ABB RAPID module: Module1.mod

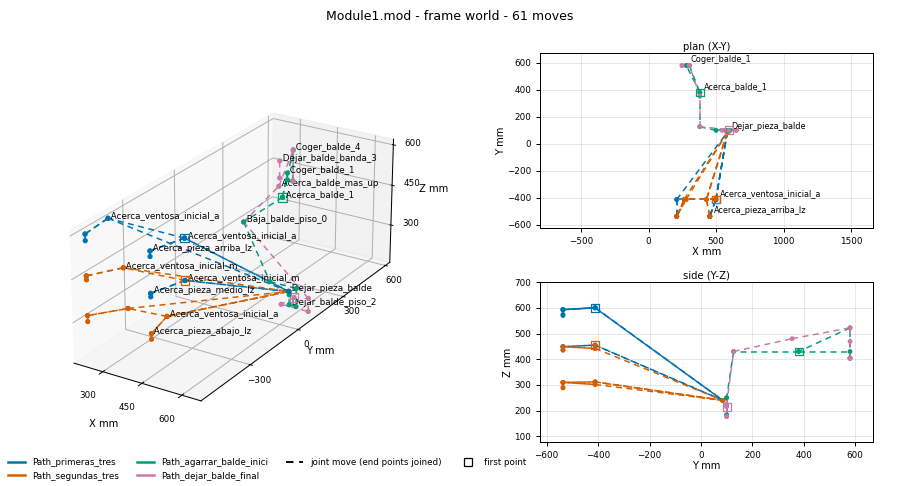
[picture p0: tool path of Module1.mod in frame world, 61 of 62 moves have a stored position in this frame; points joined in program order, loops and branches not executed]
MODULE Module1
    CONST jointtarget JointTarget_1:=[[0,0,0,0,0,0],[9E+09,9E+09,9E+09,9E+09,9E+09,9E+09]];
    CONST robtarget Acerca_balde:=[[100,70,-180],[1,0,0,0],[0,0,-1,0],[9E+09,9E+09,9E+09,9E+09,9E+09,9E+09]];
    CONST robtarget negativo_x_mundo_balde:=[[-100,170,-180],[1,0,0,0],[0,0,-1,0],[9E+09,9E+09,9E+09,9E+09,9E+09,9E+09]];
    CONST robtarget negativo_z_mundo_balde:=[[-100.000020105,169.99997294,-154.000005055],[1,0.000000007,-0.00000001,0.000000008],[0,0,-1,0],[9E+09,9E+09,9E+09,9E+09,9E+09,9E+09]];
    CONST robtarget positivo_x_mundo_balde:=[[-100,147,-154],[1,0,0,0],[0,0,-1,0],[9E+09,9E+09,9E+09,9E+09,9E+09,9E+09]];
    CONST robtarget positivo_z_mundo_balde:=[[-100,147,-217],[1,0,0,0],[0,0,-1,0],[9E+09,9E+09,9E+09,9E+09,9E+09,9E+09]];
    CONST robtarget Baja_balde_piso_0:=[[353,70,-180],[1,0,0,0],[0,0,-1,0],[9E+09,9E+09,9E+09,9E+09,9E+09,9E+09]];
    CONST robtarget Baja_balde_piso_1:=[[380,-50,0],[1,0,0,0],[0,0,-1,0],[9E+09,9E+09,9E+09,9E+09,9E+09,9E+09]];
    CONST robtarget Baja_balde_piso_2:=[[380.0000088,-152.999992201,0.000005224],[1,0.000000008,0,-0.000000022],[0,-1,-2,0],[9E+09,9E+09,9E+09,9E+09,9E+09,9E+09]];
    CONST robtarget negativo_z_balde_piso:=[[380,-153,67],[1,0,0,0],[0,0,0,0],[9E+09,9E+09,9E+09,9E+09,9E+09,9E+09]];
    CONST robtarget negativo_x_gancho_mundo_piso:=[[380,-126,67],[1,0,0,0],[0,0,-1,0],[9E+09,9E+09,9E+09,9E+09,9E+09,9E+09]];
    CONST robtarget positivo_z_gancho_mundo_piso:=[[380,-126,30],[1,0,0,0],[0,0,-1,0],[9E+09,9E+09,9E+09,9E+09,9E+09,9E+09]];
    CONST robtarget Diagonal_bajar_manija:=[[380,-185,60],[1,0,0,0],[0,0,-1,0],[9E+09,9E+09,9E+09,9E+09,9E+09,9E+09]];
    CONST robtarget Acerca_ventosa_inicial_arriba_Iz:=[[100,200,112],[1,0,0,0],[-1,-2,0,0],[9E+09,9E+09,9E+09,9E+09,9E+09,9E+09]];
    CONST robtarget negativ_y_vento_work_arriba_Iz:=[[145,75,122],[1,0,0,0],[-1,-2,0,0],[9E+09,9E+09,9E+09,9E+09,9E+09,9E+09]];
    CONST robtarget Dejar_pieza_en_balde:=[[-19.141559839,402.142254512,270],[1,0,0,-0.000000001],[-1,-2,0,0],[9E+09,9E+09,9E+09,9E+09,9E+09,9E+09]];
    CONST robtarget Acerca_ventosa_inicial_arriba_De:=[[390,200,111],[1,0,0,0],[-1,-2,0,0],[9E+09,9E+09,9E+09,9E+09,9E+09,9E+09]];
    CONST robtarget negativ_y_vento_work_arriba_De:=[[390,75,119],[1,0,0,0],[-1,-2,0,0],[9E+09,9E+09,9E+09,9E+09,9E+09,9E+09]];
    CONST robtarget Acerca_ventosa_inicial_medio_Iz:=[[100,200,257],[1,0,0,0],[-1,-2,0,0],[9E+09,9E+09,9E+09,9E+09,9E+09,9E+09]];
    CONST robtarget negativ_y_vento_work_medio_Iz:=[[145,75,258],[1,0,0,0],[-1,-2,0,0],[9E+09,9E+09,9E+09,9E+09,9E+09,9E+09]];
    CONST robtarget Agarrar_balde_again_ini:=[[380,-145,35],[1,0,0,0],[0,0,-1,0],[9E+09,9E+09,9E+09,9E+09,9E+09,9E+09]];
    CONST robtarget Agarrar_balde_again_z_nega_mun:=[[380.0000022,-95.000012886,73.00000505],[1,0.000000008,0,-0.000000022],[0,0,-2,0],[9E+09,9E+09,9E+09,9E+09,9E+09,9E+09]];
    CONST robtarget Agarrar_balde_again_x_posi_mun:=[[380,-200,73],[1,0,0,0],[0,0,-1,0],[9E+09,9E+09,9E+09,9E+09,9E+09,9E+09]];
    CONST robtarget Agarrar_balde_again_z_posi_mun:=[[380,-200,25],[1,0,0,0],[0,0,-1,0],[9E+09,9E+09,9E+09,9E+09,9E+09,9E+09]];
    CONST robtarget negativo_z_mundo_balde_dejar:=[[-100,147,-154],[1,0,0,0],[0,0,-1,0],[9E+09,9E+09,9E+09,9E+09,9E+09,9E+09]];
    CONST robtarget negativo_x_mundo_balde_dejar:=[[-100,202,-154],[1,0,0,0],[0,0,-1,0],[9E+09,9E+09,9E+09,9E+09,9E+09,9E+09]];
    CONST robtarget positivo_z_mundo_balde_dejar_H:=[[-100,202,-219],[1,0,0,0],[0,0,-1,0],[9E+09,9E+09,9E+09,9E+09,9E+09,9E+09]];
    CONST robtarget Acerca_ventosa_inicial_medio_De:=[[335,200,270],[1,0,0,0],[-1,-2,0,0],[9E+09,9E+09,9E+09,9E+09,9E+09,9E+09]];
    CONST robtarget negativ_y_vento_work_medio_De:=[[390,75,270],[1,0,0,0],[-1,-2,0,0],[9E+09,9E+09,9E+09,9E+09,9E+09,9E+09]];
    CONST robtarget Punto_intermedio_abajo_Iz:=[[170,200,300],[1,0,0,0],[-1,-2,0,0],[9E+09,9E+09,9E+09,9E+09,9E+09,9E+09]];
    CONST robtarget Acerca_ventosa_inicial_abajo_Iz:=[[170,200,400],[1,0,0,0],[-1,-2,0,0],[9E+09,9E+09,9E+09,9E+09,9E+09,9E+09]];
    CONST robtarget negativ_y_vento_work_abajo_Iz_3:=[[145,75,412],[1,0,0,0],[-1,-2,0,0],[9E+09,9E+09,9E+09,9E+09,9E+09,9E+09]];
    CONST robtarget Acerca_ventosa_inicial_abajo_De:=[[320,200,410],[1,0,0,0],[-1,-2,0,0],[9E+09,9E+09,9E+09,9E+09,9E+09,9E+09]];
    CONST robtarget negativ_y_vento_work_abajo_De_3:=[[390,75,412],[1,0,0,0],[-1,-2,0,0],[9E+09,9E+09,9E+09,9E+09,9E+09,9E+09]];
    CONST robtarget Acerca_pieza_arriba_Iz:=[[145,75,119],[1,0,0,0],[-1,-2,0,0],[9E+09,9E+09,9E+09,9E+09,9E+09,9E+09]];
    CONST robtarget Tomar_pieza_arriba_De:=[[390,75,141.8],[1,0,0,0],[-1,-2,0,0],[9E+09,9E+09,9E+09,9E+09,9E+09,9E+09]];
    CONST robtarget Tomar_pieza_medio_Iz:=[[145,75,275],[1,0,0,0],[-1,-2,0,0],[9E+09,9E+09,9E+09,9E+09,9E+09,9E+09]];
    CONST robtarget Tomar_pieza_arriba_Iz:=[[145,75,137.7],[1,0,0,0],[-1,-2,0,0],[9E+09,9E+09,9E+09,9E+09,9E+09,9E+09]];
    CONST robtarget Dejar_pieza_balde:=[[20,-15,-240],[1,0,0,0],[0,-1,0,0],[9E+09,9E+09,9E+09,9E+09,9E+09,9E+09]];
    CONST robtarget Acerca_pieza_arriba_De:=[[390,75,119],[1,0,0,0],[-1,-2,0,0],[9E+09,9E+09,9E+09,9E+09,9E+09,9E+09]];
    CONST robtarget Acerca_pieza_medio_Iz:=[[145,75,263],[1,0,0,0],[-1,-2,0,0],[9E+09,9E+09,9E+09,9E+09,9E+09,9E+09]];
    CONST robtarget Acerca_balde_mas_up:=[[125,70,-230],[1,0,0,0],[0,0,-1,0],[9E+09,9E+09,9E+09,9E+09,9E+09,9E+09]];
    CONST robtarget Tomar_pieza_medio_De:=[[390,75,276.9],[1,0,0,0],[-1,-2,0,0],[9E+09,9E+09,9E+09,9E+09,9E+09,9E+09]];
    CONST robtarget Tomar_pieza_abajo_De:=[[390,75,423.2],[1,0,0,0],[-1,-2,0,0],[9E+09,9E+09,9E+09,9E+09,9E+09,9E+09]];
    CONST robtarget Acerca_pieza_medio_De:=[[390,75,263],[1,0,0,0],[-1,-2,0,0],[9E+09,9E+09,9E+09,9E+09,9E+09,9E+09]];
    CONST robtarget Tomar_pieza_abajo_Iz:=[[145,75,421.6],[1,0,0,0],[-1,-2,0,0],[9E+09,9E+09,9E+09,9E+09,9E+09,9E+09]];
    CONST robtarget Acerca_pieza_abajo_Iz:=[[145,75,402],[1,0,0,0],[-1,-2,0,0],[9E+09,9E+09,9E+09,9E+09,9E+09,9E+09]];
    CONST robtarget Acerca_pieza_abajo_De:=[[390,75,402],[1,0,0,0],[-1,-2,0,0],[9E+09,9E+09,9E+09,9E+09,9E+09,9E+09]];
    CONST robtarget Acerca_balde_1:=[[100,70,-180],[1,0,0,0],[0,0,-1,0],[9E+09,9E+09,9E+09,9E+09,9E+09,9E+09]];
    CONST robtarget Coger_balde_1:=[[-100,170,-180],[1,0,0,0],[0,0,-1,0],[9E+09,9E+09,9E+09,9E+09,9E+09,9E+09]];
    CONST robtarget Coger_balde_2:=[[-100.000020105,169.99997294,-154.000005055],[1,0.000000007,-0.00000001,0.000000008],[0,0,-1,0],[9E+09,9E+09,9E+09,9E+09,9E+09,9E+09]];
    CONST robtarget Coger_balde_3:=[[-100,147,-154],[1,0,0,0],[0,0,-1,0],[9E+09,9E+09,9E+09,9E+09,9E+09,9E+09]];
    CONST robtarget Coger_balde_4:=[[-100,147,-272],[1,0,0,0],[0,0,-1,0],[9E+09,9E+09,9E+09,9E+09,9E+09,9E+09]];
    CONST robtarget Dejar_balde_piso_1:=[[380,-153,67],[1,0,0,0],[0,0,0,0],[9E+09,9E+09,9E+09,9E+09,9E+09,9E+09]];
    CONST robtarget Dejar_balde_piso_2:=[[380,-126,67],[1,0,0,0],[0,0,-1,0],[9E+09,9E+09,9E+09,9E+09,9E+09,9E+09]];
    CONST robtarget Dejar_balde_piso_3:=[[380,-126,30],[1,0,0,0],[0,0,-1,0],[9E+09,9E+09,9E+09,9E+09,9E+09,9E+09]];
    CONST robtarget Dejar_balde_banda_1:=[[-100,147,-154],[1,0,0,0],[0,0,-1,0],[9E+09,9E+09,9E+09,9E+09,9E+09,9E+09]];
    CONST robtarget Dejar_balde_banda_2:=[[-100,202,-154],[1,0,0,0],[0,0,-1,0],[9E+09,9E+09,9E+09,9E+09,9E+09,9E+09]];
    CONST robtarget Dejar_balde_banda_3:=[[-100,202,-219],[1,0,0,0],[0,0,-1,0],[9E+09,9E+09,9E+09,9E+09,9E+09,9E+09]];
    CONST robtarget Dejar_pieza_balde_2:=[[20,-15,-240],[0.707106781,0,0.707106781,0],[0,-1,-1,0],[9E+09,9E+09,9E+09,9E+09,9E+09,9E+09]];
    !***********************************************************
    !
    ! Módulo:  Module1
    !
    ! Descripción:
    !   <Introduzca la descripción aquí>
    !
    ! Autor: ASUS
    !
    ! Versión: 1.0
    !
    !***********************************************************


    !***********************************************************
    !
    ! Procedimiento Main
    !
    !   Este es el punto de entrada de su programa
    !
    !***********************************************************
    PROC main()
        !Añada aquí su código

        Home; !Inicio en Home
        Path_agarrar_balde_inicio;   !Coger balde de la banda y ponerlo en el piso
        Path_primeras_tres;   !Agarrar_primeras_tres_piezas
        !Path_segundas_tres;  !Agarrar_segundas_tres_piezas
        Path_dejar_balde_final;  !Dejar balde otra vez en la banda
        Home; !Finalizacion en Home

    ENDPROC

    PROC Home()
        MoveAbsJ JointTarget_1,v300,z100,Gancho\WObj:=Workobject_banda_gancho;
    ENDPROC
    PROC Path_primeras_tres()
        SetDO DO_01,0;
        SetDO DO_02,0;
        MoveJ Acerca_ventosa_inicial_arriba_Iz,v100,z100,Ventosa\WObj:=Workobject_Ventosa_Estante;
        SetDO DO_01,0;
        WaitTime 1;
        SetDO DO_02,1;
        WaitTime 1;
        MoveJ Acerca_pieza_arriba_Iz,v100,z100,Ventosa\WObj:=Workobject_Ventosa_Estante;
        MoveJ Tomar_pieza_arriba_Iz,v30,z100,Ventosa\WObj:=Workobject_Ventosa_Estante;
        MoveJ Acerca_pieza_arriba_Iz,v100,z100,Ventosa\WObj:=Workobject_Ventosa_Estante;
        MoveJ Acerca_ventosa_inicial_arriba_Iz,v100,z100,Ventosa\WObj:=Workobject_Ventosa_Estante;
        MoveJ Dejar_pieza_balde,v100,z100,Ventosa\WObj:=Workobject_Dejar_pieza_balde;
        WaitTime 1;
        SetDO DO_02,0;
        WaitTime 1;
        SetDO DO_01,1;
        WaitTime 1;
        MoveJ Acerca_ventosa_inicial_arriba_Iz,v100,z100,Ventosa\WObj:=Workobject_Ventosa_Estante;
        MoveJ Acerca_ventosa_inicial_arriba_De,v100,z100,Ventosa\WObj:=Workobject_Ventosa_Estante;
        WaitTime 1;
        SetDO DO_01,0;
        WaitTime 1;
        SetDO DO_02,1;
        WaitTime 1;
        MoveJ Acerca_pieza_arriba_De,v100,z100,Ventosa\WObj:=Workobject_Ventosa_Estante;
        MoveJ Tomar_pieza_arriba_De,v30,z100,Ventosa\WObj:=Workobject_Ventosa_Estante;
        MoveJ Acerca_pieza_arriba_De,v100,z100,Ventosa\WObj:=Workobject_Ventosa_Estante;
        MoveJ Acerca_ventosa_inicial_arriba_De,v100,z100,Ventosa\WObj:=Workobject_Ventosa_Estante;
        MoveJ Dejar_pieza_balde,v100,z100,Ventosa\WObj:=Workobject_Dejar_pieza_balde;
        WaitTime 1;
        SetDO DO_02,0;
        WaitTime 1;
        SetDO DO_01,1;
        WaitTime 1;
        MoveJ Acerca_ventosa_inicial_medio_Iz,v100,z100,Ventosa\WObj:=Workobject_Ventosa_Estante;
        WaitTime 1;
        SetDO DO_01,0;
        WaitTime 1;
        SetDO DO_02,1;
        WaitTime 1;
        MoveJ Acerca_pieza_medio_Iz,v100,z100,Ventosa\WObj:=Workobject_Ventosa_Estante;
        MoveJ Tomar_pieza_medio_Iz,v30,z100,Ventosa\WObj:=Workobject_Ventosa_Estante;
        MoveJ Acerca_pieza_medio_Iz,v100,z100,Ventosa\WObj:=Workobject_Ventosa_Estante;
        MoveJ Acerca_ventosa_inicial_medio_Iz,v100,z100,Ventosa\WObj:=Workobject_Ventosa_Estante;
        MoveJ Dejar_pieza_balde,v100,z100,Ventosa\WObj:=Workobject_Dejar_pieza_balde;
        WaitTime 1;
        SetDO DO_02,0;
        WaitTime 1;
        SetDO DO_01,1;
        WaitTime 1;
        SetDO DO_01,0;
        WaitTime 1;
    ENDPROC

    PROC Path_segundas_tres()
        MoveJ Acerca_ventosa_inicial_medio_Iz,v100,z100,Ventosa\WObj:=Workobject_Ventosa_Estante;
        MoveJ Acerca_ventosa_inicial_medio_De,v100,z100,Ventosa\WObj:=Workobject_Ventosa_Estante;
        WaitTime 1;
        SetDO DO_01,0;
        WaitTime 1;
        SetDO DO_02,1;
        WaitTime 1;
        MoveJ Acerca_pieza_medio_De,v100,z100,Ventosa\WObj:=Workobject_Ventosa_Estante;
        MoveJ Tomar_pieza_medio_De,v30,z100,Ventosa\WObj:=Workobject_Ventosa_Estante;
        MoveJ Acerca_pieza_medio_De,v100,z100,Ventosa\WObj:=Workobject_Ventosa_Estante;
        MoveJ Acerca_ventosa_inicial_medio_De,v100,z100,Ventosa\WObj:=Workobject_Ventosa_Estante;
        MoveJ Dejar_pieza_balde_2,v1000,z100,Ventosa\WObj:=Workobject_Dejar_pieza_balde_2;
        WaitTime 1;
        SetDO DO_02,0;
        WaitTime 1;
        SetDO DO_01,1;
        WaitTime 1;
        MoveJ Acerca_ventosa_inicial_abajo_Iz,v100,z100,Ventosa\WObj:=Workobject_Ventosa_Estante;
        WaitTime 1;
        SetDO DO_01,0;
        WaitTime 1;
        SetDO DO_02,1;
        WaitTime 1;
        MoveJ Acerca_pieza_abajo_Iz,v100,z100,Ventosa\WObj:=Workobject_Ventosa_Estante;
        MoveJ Tomar_pieza_abajo_Iz,v30,z100,Ventosa\WObj:=Workobject_Ventosa_Estante;
        MoveJ Acerca_pieza_abajo_Iz,v100,z100,Ventosa\WObj:=Workobject_Ventosa_Estante;
        MoveJ Acerca_ventosa_inicial_abajo_Iz,v100,z100,Ventosa\WObj:=Workobject_Ventosa_Estante;
        MoveJ Dejar_pieza_balde_2,v1000,z100,Ventosa\WObj:=Workobject_Dejar_pieza_balde_2;
        WaitTime 1;
        SetDO DO_02,0;
        WaitTime 1;
        SetDO DO_01,1;
        WaitTime 1;
        MoveJ Acerca_ventosa_inicial_abajo_Iz,v100,z100,Ventosa\WObj:=Workobject_Ventosa_Estante;
        MoveJ Acerca_ventosa_inicial_abajo_De,v100,z100,Ventosa\WObj:=Workobject_Ventosa_Estante;
        WaitTime 1;
        SetDO DO_01,0;
        WaitTime 1;
        SetDO DO_02,1;
        WaitTime 1;
        MoveJ Acerca_pieza_abajo_De,v100,z100,Ventosa\WObj:=Workobject_Ventosa_Estante;
        MoveJ Tomar_pieza_abajo_De,v30,z100,Ventosa\WObj:=Workobject_Ventosa_Estante;
        MoveJ Acerca_pieza_abajo_De,v100,z100,Ventosa\WObj:=Workobject_Ventosa_Estante;
        MoveJ Acerca_ventosa_inicial_abajo_De,v100,z100,Ventosa\WObj:=Workobject_Ventosa_Estante;
        MoveJ Dejar_pieza_balde_2,v1000,z100,Ventosa\WObj:=Workobject_Dejar_pieza_balde_2;
        WaitTime 1;
        SetDO DO_02,0;
        WaitTime 1;
        SetDO DO_01,1;
        WaitTime 1;
        SetDO DO_01,0;
        WaitTime 1;
    ENDPROC

    PROC Path_agarrar_balde_inicio()
        WaitDI DI_01,1;
        MoveJ Acerca_balde_1,v50,z100,Gancho\WObj:=Workobject_banda_gancho;
        MoveJ Coger_balde_1,v100,z100,Gancho\WObj:=Workobject_banda_gancho;
        MoveJ Coger_balde_2,v100,z100,Gancho\WObj:=Workobject_banda_gancho;
        MoveJ Coger_balde_3,v50,z100,Gancho\WObj:=Workobject_banda_gancho;
        MoveJ Coger_balde_4,v50,z100,Gancho\WObj:=Workobject_banda_gancho;
        MoveJ Acerca_balde_1,v50,z100,Gancho\WObj:=Workobject_banda_gancho;
        MoveJ Baja_balde_piso_0,v50,z100,Gancho\WObj:=Workobject_banda_gancho;
        MoveJ Baja_balde_piso_1,v50,z100,Gancho\WObj:=Workobject_banda_gancho;
        MoveJ Baja_balde_piso_2,v50,z100,Gancho\WObj:=Workobject_banda_gancho;
        MoveJ Dejar_balde_piso_1,v50,z100,Gancho\WObj:=Workobject_banda_gancho;
        MoveJ Dejar_balde_piso_2,v100,z100,Gancho\WObj:=Workobject_banda_gancho;
        MoveJ Dejar_balde_piso_3,v100,z100,Gancho\WObj:=Workobject_banda_gancho;
    ENDPROC
    PROC Path_dejar_balde_final()
        MoveJ Agarrar_balde_again_ini,v50,z100,Gancho\WObj:=Workobject_banda_gancho;
        MoveJ Agarrar_balde_again_z_nega_mun,v50,z100,Gancho\WObj:=Workobject_banda_gancho;
        MoveJ Agarrar_balde_again_x_posi_mun,v50,z100,Gancho\WObj:=Workobject_banda_gancho;
        MoveJ Agarrar_balde_again_z_posi_mun,v50,z100,Gancho\WObj:=Workobject_banda_gancho;
        MoveJ Baja_balde_piso_0,v50,z100,Gancho\WObj:=Workobject_banda_gancho;
        MoveJ Acerca_balde_mas_up,v50,z100,Gancho\WObj:=Workobject_banda_gancho;
        MoveJ Coger_balde_4,v50,z100,Gancho\WObj:=Workobject_banda_gancho;
        MoveJ Dejar_balde_banda_1,v50,z100,Gancho\WObj:=Workobject_banda_gancho;
        MoveJ Dejar_balde_banda_2,v50,z100,Gancho\WObj:=Workobject_banda_gancho;
        MoveJ Dejar_balde_banda_3,v50,z100,Gancho\WObj:=Workobject_banda_gancho;
    ENDPROC
ENDMODULE
